# EPICS substitutions: iocs/newportIOC/iocBoot/iocNewport/MM3000.substitutions
file "$(MOTOR)/db/motor.db"
{
pattern
{P,         N,      M,      DTYP,    C,  S,  DESC,          EGU,      DIR,  VELO,  VBAS,  ACCL,  BDST,  BVEL,  BACC,  MRES,  PREC,  DHLM,  DLLM,  INIT}
{newport:,  1,  "m$(N)",  "MM3000",  0,  0,  "motor $(N)",  mm,       Pos,  1,     .1,    .2,    0,     1,     .2,    5e-5,  5,     100,   -100,  ""}
{newport:,  2,  "m$(N)",  "MM3000",  0,  1,  "motor $(N)",  mm,       Pos,  1,     .1,    .2,    0,     1,     .2,    5e-5,  5,     100,   -100,  ""}
{newport:,  3,  "m$(N)",  "MM3000",  0,  2,  "motor $(N)",  mm,       Pos,  1,     .1,    .2,    0,     1,     .2,    5e-5,  5,     100,   -100,  ""}
{newport:,  4,  "m$(N)",  "MM3000",  0,  3,  "motor $(N)",  mm,       Pos,  1,     .1,    .2,    0,     1,     .2,    5e-5,  5,     100,   -100,  ""}
}
